// TwinCAT 3 PLC project TcEasyModbus
// Title: Easy Modbus Library
// Company: https://github.com/petr-suchy
// Author: Petr Suchý
// ProjectVersion: 0.1.0.0
// ProgramVersion: 3.1.4024.0
// libraries:
//   Tc2_ModbusSrv, * (Beckhoff Automation GmbH)
//   Tc2_Standard, * (Beckhoff Automation GmbH)
//   Tc2_System, * (Beckhoff Automation GmbH)
//   Tc3_Module, * (Beckhoff Automation GmbH)
// project tree:
//   DUTs/ ST_MBusConnection.TcDUT, ST_MBusStatus.TcDUT
//   / PlcTask.TcTTO
//   POUs/ FB_MBusFunc.TcPOU, FB_MBusReadInputRegs.TcPOU, FB_MBusReadInputs.TcPOU, FB_MBusWriteCoils.TcPOU, FB_MBusWriteHoldingRegs.TcPOU, MAIN.TcPOU
//   Version/ Global_Version.TcGVL
// real-time tasks:
//   TASK PlcTask: cycle T#10ms, priority 20, ADS port 350

CONFIGURATION TcEasyModbus
    RESOURCE PLC ON TwinCAT3
        TASK PlcTask(INTERVAL := T#10ms, PRIORITY := 20);
        PROGRAM MAIN WITH PlcTask : MAIN;
    END_RESOURCE
END_CONFIGURATION

// ---- DUTs/ST_MBusConnection.TcDUT
TYPE ST_MBusConnection :
STRUCT
    sIPAddr       	: STRING(15);
    nTCPPort      	: UINT := MODBUS_TCP_PORT;
    nUnitID       	: BYTE := 16#FF;
	tTimeout      	: TIME := T#5S;
END_STRUCT
END_TYPE

// ---- DUTs/ST_MBusStatus.TcDUT
TYPE ST_MBusStatus :
STRUCT
	bStatusOk	: BOOL;
    bBusy		: BOOL;
    bError		: BOOL;
    nErrId		: UDINT;
END_STRUCT
END_TYPE

// ---- Version/Global_Version.TcGVL
{attribute 'TcGenerated'}
{attribute 'no-analysis'}
{attribute 'linkalways'}
// This function has been automatically generated from the project information.
VAR_GLOBAL CONSTANT
	{attribute 'const_non_replaced'}
	stLibVersion_Easy_Modbus_Library : ST_LibVersion := (iMajor := 0, iMinor := 1, iBuild := 0, iRevision := 0, nFlags := 0, sVersion := '0.1.0.0');
END_VAR

// ---- POUs/MAIN.TcPOU
PROGRAM MAIN
VAR
END_VAR

END_PROGRAM

// ---- POUs/FB_MBusFunc.TcPOU
FUNCTION_BLOCK ABSTRACT FB_MBusFunc
VAR_INPUT
	stMBusConnection	: REFERENCE TO ST_MBusConnection;
	bEnable				: BOOL;
END_VAR
VAR_OUTPUT
	bStatusOk			: BOOL;
    bBusy				: BOOL;
    bError				: BOOL;
    nErrId				: UDINT;
END_VAR
VAR
	fbRunRTrig			: R_TRIG;
	fbResetFTrig		: F_TRIG;
	eReadState			: (WAIT, TRIGGER, CALLING, ERROR);
	stMBusStatus		: ST_MBusStatus;
END_VAR

fbRunRTrig(CLK := bEnable);
fbResetFTrig(CLK := bEnable);

IF eReadState = WAIT AND fbRunRTrig.Q THEN
	bBusy := TRUE;
	eReadState := TRIGGER;
END_IF

IF fbResetFTrig.Q THEN
	bStatusOk := FALSE;
	bError := FALSE;
	nErrId := 0;
	ClearFBOutput();
	IF eReadState = ERROR THEN
		eReadState := WAIT;
	END_IF
END_IF

CASE eReadState OF
	WAIT:
		// Do nothing
	TRIGGER:
		ReadFBInput();
		TriggerMBFunc();
		eReadState := CALLING;
		
	CALLING:
		IF NOT stMBusStatus.bBusy AND NOT stMBusStatus.bError THEN
			IF bEnable THEN
				bStatusOk := TRUE;
				WriteFBOutput();
				eReadState := TRIGGER;
			ELSE
				bBusy := FALSE;
				eReadState := WAIT;
			END_IF
		END_IF
		IF stMBusStatus.bError THEN
			bBusy := FALSE;
			IF bEnable THEN
				bStatusOk := FALSE;
				bError := TRUE;
				nErrId := stMBusStatus.nErrId;
				eReadState := ERROR;
			ELSE
				eReadState := WAIT;
			END_IF
		END_IF
		CallMBFunc();
		
	ERROR:
		// Do nothing
END_CASE

METHOD PROTECTED ABSTRACT CallMBFunc
VAR_INPUT
END_VAR
END_METHOD

METHOD PROTECTED ABSTRACT ClearFBOutput
VAR_INPUT
END_VAR
END_METHOD

METHOD PROTECTED ABSTRACT ReadFBInput
VAR_INPUT
END_VAR
END_METHOD

METHOD PROTECTED ABSTRACT TriggerMBFunc
VAR_INPUT
END_VAR
END_METHOD

METHOD PROTECTED ABSTRACT WriteFBOutput
VAR_INPUT
END_VAR
END_METHOD

END_FUNCTION_BLOCK

// ---- POUs/FB_MBusReadInputRegs.TcPOU
FUNCTION_BLOCK FB_MBusReadInputRegs EXTENDS FB_MBusFunc
VAR_INPUT
	nNumOfInputRegs		: WORD;
	nStartAddr			: WORD;
END_VAR
VAR_OUTPUT
	nInputReg0			: INT;
	nInputReg1			: INT;
	nInputReg2			: INT;
	nInputReg3			: INT;
	nInputReg4			: INT;
	nInputReg5			: INT;
	nInputReg6			: INT;
	nInputReg7			: INT;
END_VAR
VAR
	fbMBReadInputRegs	: FB_MBReadInputRegs;
	aReadBuffer			: ARRAY[0..7] OF INT;
END_VAR

SUPER^();

METHOD PROTECTED  CallMBFunc
VAR_INPUT
END_VAR
fbMBReadInputRegs(
	bExecute := FALSE,
	bBusy=> stMBusStatus.bBusy, 
	bError=> stMBusStatus.bError, 
	nErrId=> stMBusStatus.nErrId
);
END_METHOD

METHOD PROTECTED  ClearFBOutput
VAR_INPUT
END_VAR
nInputReg0 := 0;
nInputReg1 := 0;
nInputReg2 := 0;
nInputReg3 := 0;
nInputReg4 := 0;
nInputReg5 := 0;
nInputReg6 := 0;
nInputReg7 := 0;
END_METHOD

METHOD PROTECTED  ReadFBInput
VAR_INPUT
END_VAR
// Do nothing
END_METHOD

METHOD PROTECTED  TriggerMBFunc
VAR_INPUT
END_VAR
fbMBReadInputRegs(
	sIPAddr:= stMBUSConnection.sIPAddr, 
	nTCPPort:= stMBUSConnection.nTCPPort, 
	nUnitID:= stMBUSConnection.nUnitID, 
	nQuantity:= nNumOfInputRegs, 
	nMBAddr:= nStartAddr, 
	cbLength:= SIZEOF(aReadBuffer), 
	pDestAddr:= ADR(aReadBuffer), 
	bExecute:= TRUE, 
	tTimeout:= stMBUSConnection.tTimeout, 
	bBusy=> stMBusStatus.bBusy, 
	bError=> stMBusStatus.bError, 
	nErrId=> stMBusStatus.nErrId, 
	cbRead=> );
END_METHOD

METHOD PROTECTED  WriteFBOutput
VAR_INPUT
END_VAR
nInputReg0 := aReadBuffer[0];
nInputReg1 := aReadBuffer[1];
nInputReg2 := aReadBuffer[2];
nInputReg3 := aReadBuffer[3];
nInputReg4 := aReadBuffer[4];
nInputReg5 := aReadBuffer[5];
nInputReg6 := aReadBuffer[6];
nInputReg7 := aReadBuffer[7];
END_METHOD

END_FUNCTION_BLOCK

// ---- POUs/FB_MBusReadInputs.TcPOU
FUNCTION_BLOCK FB_MBusReadInputs EXTENDS FB_MBusFunc
VAR_INPUT
	nNumOfInputs	: WORD;
	nStartAddr		: WORD;
END_VAR
VAR_OUTPUT
	bInput0			: BOOL;
	bInput1			: BOOL;
	bInput2			: BOOL;
	bInput3			: BOOL;
	bInput4			: BOOL;
	bInput5			: BOOL;
	bInput6			: BOOL;
	bInput7			: BOOL;
	bInput8			: BOOL;
	bInput9			: BOOL;
	bInput10		: BOOL;
	bInput11		: BOOL;
	bInput12		: BOOL;
	bInput13		: BOOL;
	bInput14		: BOOL;
	bInput15		: BOOL;
END_VAR
VAR
	fbMBReadInputs	: FB_MBReadInputs;
	aReadBuffer		: ARRAY[0..1] OF BYTE;
END_VAR

SUPER^();

METHOD PROTECTED  CallMBFunc
VAR_INPUT
END_VAR
fbMBReadInputs(
	bExecute := FALSE,
	bBusy=> stMBusStatus.bBusy, 
	bError=> stMBusStatus.bError, 
	nErrId=> stMBusStatus.nErrId
);
END_METHOD

METHOD PROTECTED  ClearFBOutput
VAR_INPUT
END_VAR
bInput0 := FALSE;
bInput1 := FALSE;
bInput2 := FALSE;
bInput3 := FALSE;
bInput4 := FALSE;
bInput5 := FALSE;
bInput6 := FALSE;
bInput7 := FALSE;
bInput8 := FALSE;
bInput9 := FALSE;
bInput10 := FALSE;
bInput11 := FALSE;
bInput12 := FALSE;
bInput13 := FALSE;
bInput14 := FALSE;
bInput15 := FALSE;
END_METHOD

METHOD PROTECTED  ReadFBInput
VAR_INPUT
END_VAR
// Do nothing
END_METHOD

METHOD PROTECTED  TriggerMBFunc
VAR_INPUT
END_VAR
fbMBReadInputs(
	sIPAddr:= stMBUSConnection.sIPAddr, 
	nTCPPort:= stMBUSConnection.nTCPPort, 
	nUnitID:= stMBUSConnection.nUnitID, 
	nQuantity:= nNumOfInputs, 
	nMBAddr:= nStartAddr, 
	cbLength:= SIZEOF(aReadBuffer), 
	pDestAddr:= ADR(aReadBuffer), 
	bExecute:= TRUE, 
	tTimeout:= stMBUSConnection.tTimeout, 
	bBusy=> stMBusStatus.bBusy, 
	bError=> stMBusStatus.bError, 
	nErrId=> stMBusStatus.nErrId, 
	cbRead=> );
END_METHOD

METHOD PROTECTED  WriteFBOutput
VAR_INPUT
END_VAR
bInput0 := aReadBuffer[0].0;
bInput1 := aReadBuffer[0].1;
bInput2 := aReadBuffer[0].2;
bInput3 := aReadBuffer[0].3;
bInput4 := aReadBuffer[0].4;
bInput5 := aReadBuffer[0].5;
bInput6 := aReadBuffer[0].6;
bInput7 := aReadBuffer[0].7;
bInput8 := aReadBuffer[0].0;

bInput8 := aReadBuffer[1].0;
bInput9 := aReadBuffer[1].1;
bInput10 := aReadBuffer[1].2;
bInput11 := aReadBuffer[1].3;
bInput12 := aReadBuffer[1].4;
bInput13 := aReadBuffer[1].5;
bInput14 := aReadBuffer[1].6;
bInput15 := aReadBuffer[1].7;
END_METHOD

END_FUNCTION_BLOCK

// ---- POUs/FB_MBusWriteCoils.TcPOU
FUNCTION_BLOCK FB_MBusWriteCoils EXTENDS FB_MBusFunc
VAR_INPUT
	nNumOfCoils		: WORD;
	nStartAddr		: WORD;
	bCoil0			: BOOL;
	bCoil1			: BOOL;
	bCoil2			: BOOL;
	bCoil3			: BOOL;
	bCoil4			: BOOL;
	bCoil5			: BOOL;
	bCoil6			: BOOL;
	bCoil7			: BOOL;
	bCoil8			: BOOL;
	bCoil9			: BOOL;
	bCoil10			: BOOL;
	bCoil11			: BOOL;
	bCoil12			: BOOL;
	bCoil13			: BOOL;
	bCoil14			: BOOL;
	bCoil15			: BOOL;
END_VAR
VAR_OUTPUT
END_VAR
VAR
	fbMBWriteCoils	: FB_MBWriteCoils;
	aWriteBuffer	: ARRAY[0..1] OF BYTE;
END_VAR

SUPER^();

METHOD PROTECTED  CallMBFunc
VAR_INPUT
END_VAR
fbMBWriteCoils(
	bExecute := FALSE,
	bBusy=> stMBusStatus.bBusy, 
	bError=> stMBusStatus.bError, 
	nErrId=> stMBusStatus.nErrId
);
END_METHOD

METHOD PROTECTED  ClearFBOutput
VAR_INPUT
END_VAR
// Do noting
END_METHOD

METHOD PROTECTED  ReadFBInput
VAR_INPUT
END_VAR
aWriteBuffer[0].0 := bCoil0;
aWriteBuffer[0].1 := bCoil1;
aWriteBuffer[0].2 := bCoil2;
aWriteBuffer[0].3 := bCoil3;
aWriteBuffer[0].4 := bCoil4;
aWriteBuffer[0].5 := bCoil5;
aWriteBuffer[0].6 := bCoil6;
aWriteBuffer[0].7 := bCoil7;

aWriteBuffer[1].0 := bCoil8;
aWriteBuffer[1].1 := bCoil9;
aWriteBuffer[1].2 := bCoil10;
aWriteBuffer[1].3 := bCoil11;
aWriteBuffer[1].4 := bCoil12;
aWriteBuffer[1].5 := bCoil13;
aWriteBuffer[1].6 := bCoil14;
aWriteBuffer[1].7 := bCoil15;
END_METHOD

METHOD PROTECTED  TriggerMBFunc
VAR_INPUT
END_VAR
fbMBWriteCoils(
	sIPAddr:= stMBUSConnection.sIPAddr, 
	nTCPPort:= stMBUSConnection.nTCPPort, 
	nUnitID:= stMBUSConnection.nUnitID, 
	nQuantity:= nNumOfCoils, 
	nMBAddr:= nStartAddr, 
	cbLength:= SIZEOF(aWriteBuffer), 
	pSrcAddr:= ADR(aWriteBuffer), 
	bExecute:= TRUE, 
	tTimeout:= stMBUSConnection.tTimeout, 
	bBusy=> stMBusStatus.bBusy, 
	bError=> stMBusStatus.bError, 
	nErrId=> stMBusStatus.nErrId);
END_METHOD

METHOD PROTECTED  WriteFBOutput
VAR_INPUT
END_VAR
// Do nothing
END_METHOD

END_FUNCTION_BLOCK

// ---- POUs/FB_MBusWriteHoldingRegs.TcPOU
FUNCTION_BLOCK FB_MBusWriteHoldingRegs EXTENDS FB_MBusFunc
VAR_INPUT
	nNumOfHoldingRegs	: WORD;
	nStartAddr			: WORD;
	nHoldingReg0		: INT;
	nHoldingReg1		: INT;
	nHoldingReg2		: INT;
	nHoldingReg3		: INT;
	nHoldingReg4		: INT;
	nHoldingReg5		: INT;
	nHoldingReg6		: INT;
	nHoldingReg7		: INT;	
END_VAR
VAR_OUTPUT
END_VAR
VAR
	fbMBWriteRegs	: FB_MBWriteRegs;
	aWriteBuffer	: ARRAY[0..7] OF INT;
END_VAR

SUPER^();

METHOD PROTECTED  CallMBFunc
VAR_INPUT
END_VAR
fbMBWriteRegs(
	bExecute := FALSE,
	bBusy=> stMBusStatus.bBusy, 
	bError=> stMBusStatus.bError, 
	nErrId=> stMBusStatus.nErrId
);
END_METHOD

METHOD PROTECTED  ClearFBOutput
VAR_INPUT
END_VAR
// Do noting
END_METHOD

METHOD PROTECTED  ReadFBInput
VAR_INPUT
END_VAR
aWriteBuffer[0] := nHoldingReg0;
aWriteBuffer[1] := nHoldingReg1;
aWriteBuffer[2] := nHoldingReg2;
aWriteBuffer[3] := nHoldingReg3;
aWriteBuffer[4] := nHoldingReg4;
aWriteBuffer[5] := nHoldingReg5;
aWriteBuffer[6] := nHoldingReg6;
aWriteBuffer[7] := nHoldingReg7;
END_METHOD

METHOD PROTECTED  TriggerMBFunc
VAR_INPUT
END_VAR
fbMBWriteRegs(
	sIPAddr:= stMBUSConnection.sIPAddr, 
	nTCPPort:= stMBUSConnection.nTCPPort, 
	nUnitID:= stMBUSConnection.nUnitID, 
	nQuantity:= nNumOfHoldingRegs, 
	nMBAddr:= nStartAddr, 
	cbLength:= SIZEOF(aWriteBuffer), 
	pSrcAddr:= ADR(aWriteBuffer), 
	bExecute:= TRUE, 
	tTimeout:= stMBUSConnection.tTimeout, 
	bBusy=> stMBusStatus.bBusy, 
	bError=> stMBusStatus.bError, 
	nErrId=> stMBusStatus.nErrId);
END_METHOD

METHOD PROTECTED  WriteFBOutput
VAR_INPUT
END_VAR
// Do nothing
END_METHOD

END_FUNCTION_BLOCK
